PROGRAM P_PLC_Diagnostics
VAR
	//FB
	fbCheckLicense	:	FB_CheckLicense;
	fbGetSystemId	:	FB_GetSystemId;
	//Variables
	xGetSystemId: BOOL;
END_VAR

END_PROGRAM

(* stored: Version 1.1.0.1, ProductVersion 3.1.4022.12
   POU P_PLC_Diagnostics: Id {102759fd-9553-4b1c-afe0-5109c46f73f2}, SpecialFunc None *)
